FUNCTION_BLOCK EVENT_ACCUMULATOR
  {SET_ATTRIBUTE(OpcUa, SERVICE)}
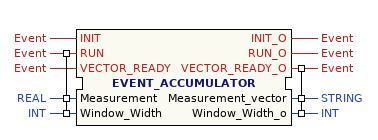
  EVENT_INPUT
    INIT;
    RUN WITH Measurement, Window_Width; {SET_ATTRIBUTE(OpcUa, Method)}
    VECTOR_READY;
  END_EVENT
  EVENT_OUTPUT
    INIT_O;
    RUN_O;
    VECTOR_READY_O WITH Measurement_vector, Window_Width_o;
  END_EVENT
  VAR_INPUT
    Measurement : REAL; {SET_ATTRIBUTE(OpcUa, Variable.RUN)}
    Window_Width : INT; {SET_ATTRIBUTE(OpcUa, Variable.RUN)}
  END_VAR
  VAR_OUTPUT
    Measurement_vector : STRING; {SET_ATTRIBUTE(OpcUa, Variable.RUN)}
    Window_Width_o : INT; {SET_ATTRIBUTE(OpcUa, Variable.RUN)}
  END_VAR
END_FUNCTION_BLOCK
